(****************************************************************
NAME:			FB_SetAxisPosition
DATA:			2017.2.16
VERSION:		1.0.0
DESCRIPTION:	FB_SetAxisPosition
HISTORY:
				2017.2.16		NEW

***************************************************************)
FUNCTION_BLOCK FB_SetMotorAxisPosition
VAR_INPUT
	//GapValueSet:LREAL:=0;
	ValueSet_LeftTop:LREAL:=0;
	ValueSet_RightTop:LREAL:=0;
	ValueSet_LeftBottom:LREAL:=0;
	ValueSet_RightBottom:LREAL:=0;
	ValueSet_LeftIn:LREAL:=0;
	ValueSet_RightIn:LREAL:=0;
	ValueSet_LeftOut:LREAL:=0;
	ValueSet_RightOut:LREAL:=0;
	Execute:BOOL;
END_VAR
VAR_OUTPUT
	FbID:DINT:=1001;
	State:DINT;
	Busy:BOOL;
	Done:BOOL;
	Error:BOOL;
	ErrorID:DINT;
END_VAR
VAR
	LeftTopMotor_MC_SetPosition: MC_SetPosition;
	RightTopMotor_MC_SetPosition: MC_SetPosition;
	LeftBottomMotor_MC_SetPosition: MC_SetPosition;
	RightBottomMotor_MC_SetPosition: MC_SetPosition;
	LeftInMotor_MC_SetPosition: MC_SetPosition;
	RightInMotor_MC_SetPosition: MC_SetPosition;
	LeftOutMotor_MC_SetPosition: MC_SetPosition;
	RightOutMotor_MC_SetPosition: MC_SetPosition;
	fb_ton: TON;
	FB_PlcEmergencyStop: FB_PlcEmergencyStop;

END_VAR

IF Execute THEN
Busy:=TRUE;
Done:=FALSE;
fb_ton(PT:=t#0.1s);
CASE State OF
	0:
		IF LeftTopMotor_MC_SetPosition.Error OR RightTopMotor_MC_SetPosition.Error
			OR LeftBottomMotor_MC_SetPosition.Error OR RightBottomMotor_MC_SetPosition.Error 
			OR LeftInMotor_MC_SetPosition.Error OR RightInMotor_MC_SetPosition.Error
			OR LeftOutMotor_MC_SetPosition.Error OR RightOutMotor_MC_SetPosition.Error THEN		(*FB Error*)
			ErrorID:=1;
			State:=99;
		ELSE
			State:=1;
		END_IF
	1:	(*Execute*)
		LeftTopMotor_MC_SetPosition.Position:=ValueSet_LeftTop;
		LeftTopMotor_MC_SetPosition.Execute:=TRUE;
		RightTopMotor_MC_SetPosition.Position:=ValueSet_RightTop;
		RightTopMotor_MC_SetPosition.Execute:=TRUE;
		LeftBottomMotor_MC_SetPosition.Position:=ValueSet_LeftBottom;
		LeftBottomMotor_MC_SetPosition.Execute:=TRUE;
		RightBottomMotor_MC_SetPosition.Position:=ValueSet_RightBottom;
		RightBottomMotor_MC_SetPosition.Execute:=TRUE;
		//
		LeftInMotor_MC_SetPosition.Position:=ValueSet_LeftIn;
		LeftInMotor_MC_SetPosition.Execute:=TRUE;
		RightInMotor_MC_SetPosition.Position:=ValueSet_RightIn;
		RightInMotor_MC_SetPosition.Execute:=TRUE;
		LeftOutMotor_MC_SetPosition.Position:=ValueSet_LeftOut;
		LeftOutMotor_MC_SetPosition.Execute:=TRUE;
		RightOutMotor_MC_SetPosition.Position:=ValueSet_RightOut;
		RightOutMotor_MC_SetPosition.Execute:=TRUE;
		A_SetPositionMC();
		fb_ton.IN:=TRUE;
		State:=2;
	2:	(*Wait*)
		A_SetPositionMC();
		IF NOT LeftTopMotor_MC_SetPosition.Done OR NOT RightTopMotor_MC_SetPosition.Done
			OR NOT LeftBottomMotor_MC_SetPosition.Done OR NOT RightBottomMotor_MC_SetPosition.Done 
			OR NOT LeftInMotor_MC_SetPosition.Done OR NOT RightInMotor_MC_SetPosition.Done
			OR NOT LeftOutMotor_MC_SetPosition.Done OR NOT RightOutMotor_MC_SetPosition.Done THEN		(*DoneÐÅºÅ²»µ½£¬¼ÌÐøµÈ´ý£¬Èç¹û³¬Ê±ÔòFB Error*)
			IF NOT fb_ton.Q THEN
				State:=2;
			ELSE
				ErrorID:=4;
				State:=99;
			END_IF
		ELSIF  LeftTopMotor_MC_SetPosition.Done AND RightTopMotor_MC_SetPosition.Done
			AND LeftBottomMotor_MC_SetPosition.Done AND RightBottomMotor_MC_SetPosition.Done 
			AND LeftInMotor_MC_SetPosition.Done AND RightInMotor_MC_SetPosition.Done
			AND LeftOutMotor_MC_SetPosition.Done AND RightOutMotor_MC_SetPosition.Done THEN		(*Done£¬×ªÏÂÒ»²½*)
			State:=88;
		ELSE
			ErrorID:=5;
			State:=99;
		END_IF
	88:
		Execute:=FALSE;
		State:=0;
		Busy:=FALSE;
		Done:=TRUE;
		Error:=FALSE;
		ErrorID:=0;
		LeftTopMotor_MC_SetPosition.Execute:=FALSE;
		RightTopMotor_MC_SetPosition.Execute:=FALSE;
		LeftBottomMotor_MC_SetPosition.Execute:=FALSE;
		RightBottomMotor_MC_SetPosition.Execute:=FALSE;
		LeftInMotor_MC_SetPosition.Execute:=FALSE;
		RightInMotor_MC_SetPosition.Execute:=FALSE;
		LeftOutMotor_MC_SetPosition.Execute:=FALSE;
		RightOutMotor_MC_SetPosition.Execute:=FALSE;
		fb_ton.IN:=FALSE;
	99:
		Execute:=FALSE;
		State:=99;
		Busy:=FALSE;
		Done:=FALSE;
		Error:=TRUE;
		LeftTopMotor_MC_SetPosition.Execute:=FALSE;
		RightTopMotor_MC_SetPosition.Execute:=FALSE;
		LeftBottomMotor_MC_SetPosition.Execute:=FALSE;
		RightBottomMotor_MC_SetPosition.Execute:=FALSE;
		LeftInMotor_MC_SetPosition.Execute:=FALSE;
		RightInMotor_MC_SetPosition.Execute:=FALSE;
		LeftOutMotor_MC_SetPosition.Execute:=FALSE;
		RightOutMotor_MC_SetPosition.Execute:=FALSE;
		fb_ton.IN:=FALSE;
	-100:
		FB_PlcEmergencyStop();
		Execute:=FALSE;
		State:=-100;
		Busy:=FALSE;
		Done:=FALSE;
		Error:=TRUE;
		LeftTopMotor_MC_SetPosition.Execute:=FALSE;
		RightTopMotor_MC_SetPosition.Execute:=FALSE;
		LeftBottomMotor_MC_SetPosition.Execute:=FALSE;
		RightBottomMotor_MC_SetPosition.Execute:=FALSE;
		
		LeftInMotor_MC_SetPosition.Execute:=FALSE;
		RightInMotor_MC_SetPosition.Execute:=FALSE;
		LeftOutMotor_MC_SetPosition.Execute:=FALSE;
		RightOutMotor_MC_SetPosition.Execute:=FALSE;
		fb_ton.IN:=FALSE;
END_CASE
END_IF

ACTION A_SetPositionMC:
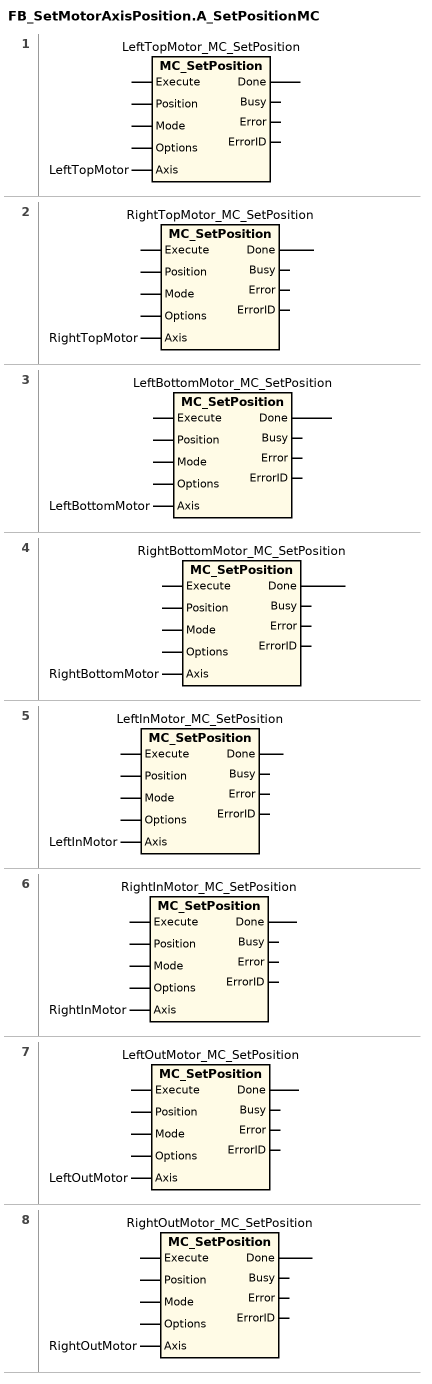
// NETWORK 1
LeftTopMotor_MC_SetPosition(Axis := LeftTopMotor); // MC_SetPosition

// NETWORK 2
RightTopMotor_MC_SetPosition(Axis := RightTopMotor); // MC_SetPosition

// NETWORK 3
LeftBottomMotor_MC_SetPosition(Axis := LeftBottomMotor); // MC_SetPosition

// NETWORK 4
RightBottomMotor_MC_SetPosition(Axis := RightBottomMotor); // MC_SetPosition

// NETWORK 5
LeftInMotor_MC_SetPosition(Axis := LeftInMotor); // MC_SetPosition

// NETWORK 6
RightInMotor_MC_SetPosition(Axis := RightInMotor); // MC_SetPosition

// NETWORK 7
LeftOutMotor_MC_SetPosition(Axis := LeftOutMotor); // MC_SetPosition

// NETWORK 8
RightOutMotor_MC_SetPosition(Axis := RightOutMotor); // MC_SetPosition
END_ACTION

END_FUNCTION_BLOCK

(* stored: Version 1.1.0.1, ProductVersion 3.1.4024.6
   POU FB_SetMotorAxisPosition: Id {7ff7f3e3-61ea-4e6e-abb0-7cca367980f1}, SpecialFunc None
   Action A_SetPositionMC: Id {4305f8a6-aed8-4378-8c07-b1e69cff0c03} *)
